// TIA Portal V17 export
// export: Created 2025-11-19T10:30:00.000Z, ExportSetting WithDefaults, DisplayName Totally Integrated Automation Portal, DisplayVersion V17
FUNCTION "FC_MotorControl" : Void   // FC10, SCL
{ S7_Optimized_Access := 'TRUE' }
AUTHOR : Engineering Team
FAMILY : Motors
NAME : Motor Control Function
VERSION : 1.0
// stored: AutoNumber true, IsIECCheckEnabled true
   VAR_INPUT
      Start : Bool;
      Stop : Bool;
      Speed_Setpoint : Real;
   END_VAR
   VAR_OUTPUT
      Motor_On : Bool;
      Current_Speed : Real;
   END_VAR
   VAR_TEMP
      temp_speed : Real;
   END_VAR
BEGIN
// Motor Control - BUGGY
// BUGS: Stop acts as Start, race condition, no emergency stop, missing speed limits, immediate stop without ramp-down, no state validation
   0.0 THEN #Motor_On := FALSE;#Motor_On = FALSE;#Motor_On = FALSE; END_IF;#Motor_On = FALSE; END_IF;#Motor_On = FALSE; END_IF;#Motor_On = FALSE; END_IF;#Motor_On = FALSE; END_IF;#Motor_On = FALSE; END_
END_FUNCTION
